Fanuc KAREL source: CHR.kl

PROGRAM T
%NOLOCKGROUP
VAR
 v0 : INTEGER
 res : STRING[40]
BEGIN
 res = CHR(v0)
END T
